Universal Robots PolyScope program: unveiling.urp

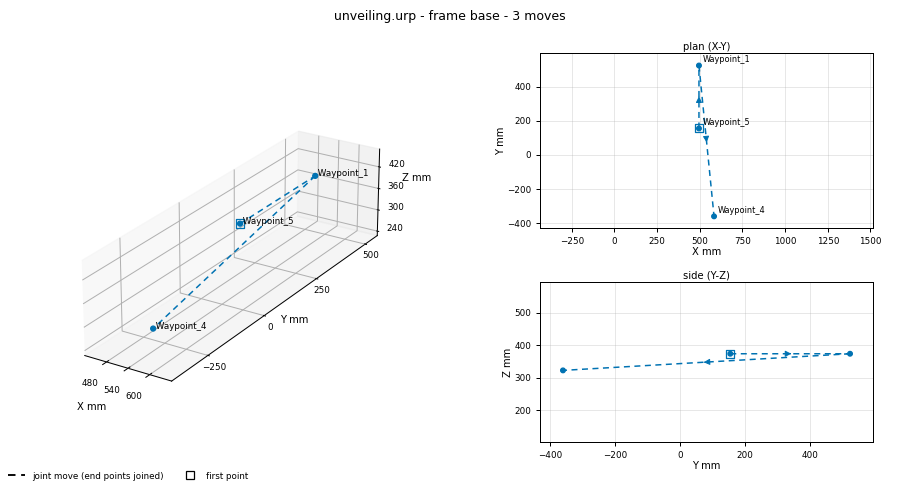
[picture p0: tool path of unveiling.urp in frame base, 3 of 3 moves have a stored position in this frame; points joined in program order, loops and branches not executed]
Program unveiling (createdIn=3.4.4.412 lastSavedIn=3.4.4.412 directory=/programs installation=default robotSerialNumber=2017356443)
Calibrated DH parameters: a=[0.000092, -0.116521, -0.182101, -0.000106, 0.000044, 0]; d=[0.089391, 255.189113, -82.629387, -172.449369, 0.094782, 0.082637]; alpha=[1.569598, 0.001603, 0.002015, 1.570234, -1.570307, 0]; deltaTheta=[-0.000017, 1.293309, -0.204843, -1.088417, 0.000036, -0.000078]
Robot Program (runOnlyOnce=true motionType=MoveJ speed=1.047198 acceleration=1.396263 useActiveTCP=false)
  URCap Gripper (Robotiq_2-Finger_Adaptive_Gripper, Robotiq Inc.) data=position = 0
    | force = 100
    | speed = 100
    | blocking = true
    | slaveIds = [9]
  MoveJ speed 60 deg/s, acceleration 80 deg/s^2 (useActiveTCP=false)
    Waypoint Waypoint_5: TCP in base x=494.971 y=154.79 z=373.805 mm, rx=-0.0574 ry=-2.3379 rz=-2.0815 rad; joints [21.23, -106.765, -76.57, -193.697, -157.06, -13.842] deg
  MoveJ speed 60 deg/s, acceleration 80 deg/s^2 (useActiveTCP=false)
    Waypoint Waypoint_1: TCP in base x=494.99 y=523.472 z=373.804 mm, rx=-0.0574 ry=-2.3379 rz=-2.0815 rad; joints [51.474, -131.209, -38.87, -198.222, -127.484, -3.125] deg
  URCap Gripper (Robotiq_2-Finger_Adaptive_Gripper, Robotiq Inc.) data=position = 100
    | force = 100
    | speed = 100
    | blocking = true
    | slaveIds = [9]
  MoveJ speed 60 deg/s, acceleration 80 deg/s^2 (useActiveTCP=false)
    Waypoint Waypoint_4: TCP in base x=583.358 y=-360.248 z=322.577 mm, rx=1.2837 ry=2.3728 rz=-0.3038 rad; joints [-20.505, -145.257, -19.814, -261.757, -74.648, -56.994] deg
  URCap Gripper (Robotiq_2-Finger_Adaptive_Gripper, Robotiq Inc.) data=position = 0
    | force = 100
    | speed = 100
    | blocking = true
    | slaveIds = [9]
